(*
SPDX-FileCopyrightText: Â© 2026 Oleksandr Tiutyk <trofimich@gmail.com>
SPDX-License-Identifier: MIT
License: https://opensource.org/license/mit
*)

(*!
<summary>Strategy for handling critical errors reported by child components.</summary>
<description>
Determines the reaction of a parent component when one of its children enters an error state.
</description>
*)

INTERFACE IChildCriticalErrorHandlingPolicy EXTENDS TOF_Core.IObject

(*!
<summary>Evaluates child error and determines the reaction to apply to the parent component.</summary>
<param name="childWithError">Child component that reported the error.</param>
<param name="handlingObject">Parent component handling the failure.</param>
<description>Returns CHILD_CRITICAL_ERROR_REACTION indicating the action to perform.</description>
*)
METHOD HandleChildCriticalError : CHILD_CRITICAL_ERROR_REACTION
VAR_INPUT
	childWithError : IChildAutomationComponent;
	handlingObject : TOF_Core.IObject;
END_VAR
END_METHOD

END_INTERFACE

(* stored: Version 1.1.0.1
   Itf IChildCriticalErrorHandlingPolicy: Id {547b6b32-97b1-4f6b-819d-55883abf3536}
   Method HandleChildCriticalError: Id {c8eef88d-a8ad-4501-b597-98276c3d795c} *)
